% RSLogix 500 project BITWISEAND_BAK059.RSS, saved by version 8.30.00.16 %
PROJECT "UNTITLED"    % processor: MicroLogix 1000 %

PROGRAM FILES
  LAD 2 "MAIN_PROG"  5 rungs
  LAD 3 "USER_FAULT"  1 rungs
  LAD 4 "HSC_INT"  1 rungs
  LAD 5 "STI_INT"  1 rungs
  LAD 6, 7, 8, 9, 10, 11, 12, 13, 14, 15, 16: only END

DATA FILES
  O0 OUTPUT  1 elements
  I1 INPUT  2 elements
  S2 STATUS  33 elements
  B3 BINARY  32 elements
  T4 TIMER  40 elements
  C5 COUNTER  32 elements
  R6 CONTROL  16 elements
  N7 INTEGER  105 elements

LADDER 2 "MAIN_PROG"
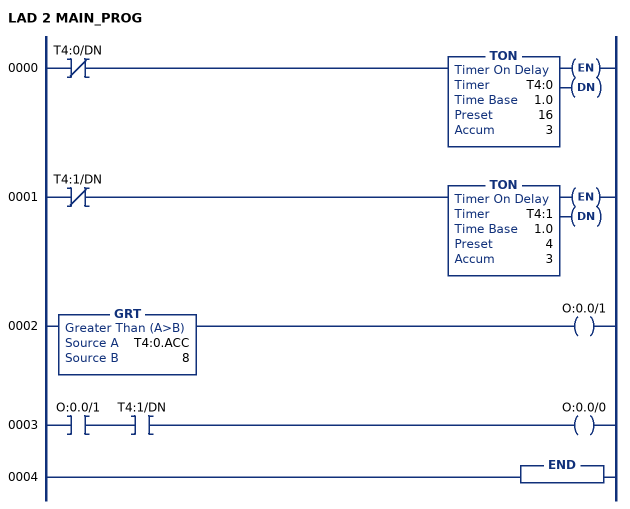
% Rung: 0 %
SOR XIO T4:0/DN TON T4:0 1.0 16 3 EOR
% Rung: 1 %
SOR XIO T4:1/DN TON T4:1 1.0 4 3 EOR
% Rung: 2 %
SOR GRT T4:0.ACC 8 OTE O:0.0/1 EOR
% Rung: 3 %
SOR XIC O:0.0/1 XIC T4:1/DN OTE O:0.0/0 EOR
% Rung: 4 %
SOR END EOR

DATA TABLE (non-zero values as saved)
DATA B3
% B3:0 % 0X000F 0X0000 0X0000 0X0000 0X0000 0X0000 0X0000 0X0000 0X0000 0X0000
DATA T4
% .PRE .ACC %
% T4:0 % 16 3
% T4:1 % 4 3
